(* IEC 61131-3 sources: mastertool-rankine-bridge/tests/indexer/fixtures/sample_export/objects/application_gvl_1__GvlDiagnosticoSintetico, 1 file *)

(* ---- declaration.st ---- *)
VAR_GLOBAL
    DG_SensorSintetico AT %IW12 : INT;
    DG_Contador : DINT;
END_VAR
